FUNCTION_BLOCK FB_StartWaterFlowState IMPLEMENTS I_State
VAR_INPUT
END_VAR
VAR_OUTPUT
END_VAR
VAR
	pMachine : POINTER TO FB_StateMachine;	
END_VAR

{warning 'Eigenschaftenimplementierung hinzufügen'}
PROPERTY Description : STRING
GET
Description := 'Opening Ventil ...';
END_GET
END_PROPERTY

{warning 'Methodenimplementierung hinzufügen'}
METHOD ErrorDetected : BOOL
VAR_IN_OUT
	errorEvents	: ST_ErrorEvents;
END_VAR
transitionToErrorState(errorEvents := errorEvents, pMachine := pMachine);
END_METHOD

//FB_Init ist immer implizit verfügbar und wird primär für die Initialisierung verwendet.
//Der Rückgabewert wird nicht ausgewertet. Für gezielte Einflussnahme können Sie
//die Methoden explizit deklarieren und darin mit dem Standard-Initialisierungscode 
//zusätzlichen Code bereitstellen. Sie können den Rückgabewert auswerten.
METHOD FB_Init: BOOL
VAR_INPUT    
	bInitRetains: BOOL; // TRUE: Die Retain-Variablen werden initialisiert (Reset warm / Reset kalt)    
	bInCopyCode: BOOL;  // TRUE: Die Instanz wird danach in den Kopiercode kopiert (Online-Change)
	pMachine : POINTER TO FB_StateMachine;
END_VAR
THIS^.pMachine := pMachine;
END_METHOD

{warning 'Methodenimplementierung hinzufügen'}
METHOD HeatIsRequested : BOOL
END_METHOD

METHOD MinWaterFlowReached : BOOL
VAR_INPUT
END_VAR
LogMessage(E_LogType.INFO, 'Ventil ist geöffnet. Durchflussmenge erreicht. Kompressor wird eingeschaltet: -> ', pMachine^.RunningState.Name);
pMachine^.pd.actor.operatingStateWaterPump := TRUE;
pMachine^.pd.actor.operatingStateIntermediateCircuitPump := TRUE;
pMachine^.pd.actor.operatingStateCompressor := TRUE;
pMachine^.SetState(pMachine^.RunningState);
END_METHOD

{warning 'Eigenschaftenimplementierung hinzufügen'}
PROPERTY Name : STRING
GET
Name := 'öffne Ventil';
END_GET
END_PROPERTY

{warning 'Eigenschaftenimplementierung hinzufügen'}
PROPERTY State : E_State
GET
State := E_State.START_WATER_FLOW;
END_GET
END_PROPERTY

{warning 'Methodenimplementierung hinzufügen'}
METHOD TargetTemperatureReached : BOOL
END_METHOD

{warning 'Methodenimplementierung hinzufügen'}
METHOD UserPressedConfirmationButton : BOOL
END_METHOD

METHOD UserPressedSwitchOffButton : BOOL
LogMessage(E_LogType.INFO, 'Aus Button wurde gedrückt -> ', pMachine^.OffState.Name);
switchWaterVentil(bOpen := FALSE, pMachine);
pMachine^.pd.actor.operatingStateCompressor := FALSE;
pMachine^.pd.actor.operatingStateWaterPump := FALSE;
pMachine^.pd.actor.operatingStateIntermediateCircuitPump := FALSE;
pMachine^.SetState(pMachine^.OffState);
END_METHOD

{warning 'Methodenimplementierung hinzufügen'}
METHOD UserPressedSwitchOnButton : BOOL
END_METHOD

{warning 'Methodenimplementierung hinzufügen'}
METHOD WaterHasCooledDown : BOOL
END_METHOD

END_FUNCTION_BLOCK

(* stored: Version 1.1.0.1
   POU FB_StartWaterFlowState: Id {d6143444-8385-4f02-ba2f-ac6faf4cc7a7}, SpecialFunc None
   Property Description: Id {85edbbf9-5af6-4227-bd92-768a7a8660f6}
   Get Get: Id {0ecedba2-0913-4b6d-b593-f32af667137c}
   Method ErrorDetected: Id {d3299433-f31e-4f24-b5b8-67543a1d3986}
   Method FB_init: Id {099a8c71-7fde-4fa0-912e-b7622d7c04c4}
   Method HeatIsRequested: Id {bc3ae7fd-9def-47d5-b24d-7241e3a96555}
   Method MinWaterFlowReached: Id {d9d57206-5755-440e-a786-4c12f144959a}
   Property Name: Id {91be18b5-b8e8-4a69-af2d-5dcef30e192b}
   Get Get: Id {cacf37de-231d-49bd-a636-7e05eac8d2eb}
   Property State: Id {f2e32701-8d1d-4e8c-b547-4a95e9c31fdf}
   Get Get: Id {60fc8015-6f48-4dec-a1a9-3520b4b3d0fe}
   Method TargetTemperatureReached: Id {183626c5-33c6-4814-93d2-48104f196c2b}
   Method UserPressedConfirmationButton: Id {15d87427-e804-4017-a28c-eb5f7982c5b9}
   Method UserPressedSwitchOffButton: Id {132cc9f9-1903-4055-8e00-9860ee28e509}
   Method UserPressedSwitchOnButton: Id {83eb9baa-fd12-4076-9a0d-d1625eff0b1b}
   Method WaterHasCooledDown: Id {810af7e9-9366-4b5e-94ea-c4a8efb0ab95} *)
